TYPE Hardware :
STRUCT
	intDriveNumber			:		INT;
	sDriveModel				:		STRING;
	sMotorModel				:		STRING;
END_STRUCT
END_TYPE

(* stored: Version 1.1.0.1, ProductVersion 3.1.4024.6
   DUT Hardware: Id {c2cb8a09-68d8-4356-8a60-e91ad42f3546} *)
